TYPE fbPistonStatus :
STRUCT
    AtHome : TIME;
    AtWork : TIME;
END_STRUCT
END_TYPE

(* stored: Version 1.1.0.1
   DUT fbPistonStatus: Id {73efb0a1-3a61-0f8f-0af2-16afb6e2118b} *)
